(* IEC 61131-3 sources: axopen.templates/axopen.template.simple/ax/src/Units/Cu10, 2 files *)

(* ---- Unit.st ---- *)
NAMESPACE axosimple.Cu10
    USING axosimple;
    USING AXOpen.Data;
    USING AXOpen.Core;
    USING System.Strings;

    ///<summary>
    /// Represents controlled units and high level task coordination.
    ///</summary>
    {S7.extern=ReadWrite}
    CLASS Unit
        EXTENDS axosimple.BaseUnit.UnitBase
        VAR PUBLIC
            ///<summary>
            /// Provide access to unit objets, that are used into sequnces.
            ///</summary>
            X  : axosimple.Cu10.UnitObjects;

            ///<summary>
            /// Ground sequence. Contains logic that brings the unit into initial state.
            ///</summary>
            Ground : axosimple.Cu10.GroundSequence;

            ///<summary>
            /// Automatic sequence. Contains logic for automatic operations of this unit.
            ///</summary>
            Auto : axosimple.Cu10.AutomatSequence;

            ///<summary>
            /// Service mode contains logic for service/manual operations.
            ///</summary>
            Service : axosimple.Cu10.ServiceMode;
        END_VAR
        ///<summary>
        /// Runs this unit.
        ///</summary>

        METHOD PUBLIC Run
            VAR_INPUT
                inParent : IAxoContext;
            END_VAR
            VAR_IN_OUT
                ///<summary>
                /// Hardware input structure
                ///</summary>
                inoInputs : axosimple.Inputs;
                ///<summary>
                /// Hardware output structure
                ///</summary>
                inoOutputs : axosimple.Outputs;
            END_VAR
            VAR_INPUT
                inGlobal : REF_TO axosimple.GlobalContextObjects;
            END_VAR
            THIS.Initialize(inParent);
            X.G := inGlobal;
            THIS.Execute(inoInputs, inoOutputs);
        END_METHOD

        ///<summary>
        ///     Exectute for this unit.
        ///     Execute runs cyclicaly you should place any call of this unit in this or underlying methods.
        ///</summary>
        METHOD PRIVATE Execute
            VAR_IN_OUT
                inoInputs : axosimple.Inputs;
                inoOutputs : axosimple.Outputs;
            END_VAR

            // Component I/O immange and management handling.
             X.C.Update(THIS, inoInputs, inoOutputs);

             // Run process data manager of this unit.
             X.PD.Run(THIS);

             // Run technology data manger of this unit.
             X.TD.Run(THIS);

            /*

                    Ground mode handling

            */

             Ground.Run(THIS, REF(X));

             // Restores other states when Ground executes
             IF (Ground.IsBusy()) THEN
                 Auto.Restore();
                 Service.Restore();
             END_IF;

             /*

                    Automatic mode handling
                    NOTE: Ground must be previously done.

             */

             Auto.IsDisabled := Ground.Status <> eAxoTaskState#Done;
             Auto.Run(THIS, REF(X));

            /*

                Service/manual mode hadnling

             */

             Service.Run(THIS, X.C);

             IF Service.IsBusy() THEN
                 Ground.Restore();
                 Auto.Restore();
             END_IF;

        END_METHOD
    END_CLASS
END_NAMESPACE

(* ---- UnitObjects.st ---- *)
NAMESPACE axosimple.Cu10

    USING axosimple;
    USING AXOpen.Data;
    USING AXOpen.Core;
    USING System.Strings;

    {S7.extern=ReadWrite}
    CLASS PUBLIC UnitObjects EXTENDS axosimple.BaseUnit.UnitObjects
        VAR PUBLIC
            ///<summary>
            /// Handles and intializes components used by this unit.
            ///</summary>
            C : axosimple.Cu10.Components;

            ///<summary>
            /// Provides access to process data manager of this unit.
            ///</summary>
            PD : axosimple.Cu10.ProcessDataManager;

            ///<summary>
            /// Provides access to technology data manager of this unit.
            ///</summary>
            TD : axosimple.Cu10.TechnologyDataManager;

            // ///<summary>
            // /// Provides access to technology settings of this unit.
            // ///</summary>
            // TS : REF_TO axosimple.Cu10.TechnologyDataExchange;

            // ///<summary>
            // /// Provides access to process setting of this unit.
            // ///</summary>
            // PS : REF_TO axosimple.Cu10.ProcessDataExchange;

            {#ix-attr:[AXOpen.Data.PersistentAttribute("Cu10")]}
            SpecialSettings :STRING[64] ;

            // https://ix-ax.github.io/AXOpen/core/docs/AXODIALOG.html#closing-a-dialog-with-external-signal
            _DL     : AXOpen.Core.AxoDialog;

            // https://ix-ax.github.io/AXOpen/core/docs/AXOALERTDIALOG.html#invoking-alerts-from-plc
            _ADL    : AXOpen.Core.AxoAlert;

            // it needs to be handle from auto or ground sequnce
            _IDL    : AXOpen.Inspectors.AxoInspectorDialog;

        END_VAR
    END_CLASS

END_NAMESPACE
